# EPICS StreamDevice protocol: epics/protocols/multi_event.proto
Terminator = LF;
ExtraInput = Ignore;
ReplyTimeout = 2500;

set_MEV {
	out "multi_event %(A)d,%(B)d,%(C)d,%(D)d";
	in;
}

get_MEV {
	out "multi_event";
	in "%s";
}
